{attribute 'qualified_only'}
{attribute 'to_string'}
TYPE eLogItemGroupID :
(	
	//None					:= 	0,
	General					:=	1,
	ACSwitchgear			:=	2,
	CoolingSystem			:=	3,
	BMS						:=	4,
	PowerStack				:=	5,
	Enclosure				:=	6,
	InternalPowerSupply		:=	7,
	Safety					:=	8,
	ZPT						:=  9,
	DClink					:= 10
) WORD := General;
END_TYPE

(* stored: Version 1.1.0.1, ProductVersion 3.1.4026.18
   DUT eLogItemGroupID: Id {214b6323-7223-4012-aeb4-5666b12e3e19} *)
